// LS Electric XG5000 project: 16-48-1
// PLC NewPLC
// module base 0 slot 0: 입출력 모듈:XBC-DR14E (DC 24V 입력 8점, 릴레이 출력 6점)

PROGRAM NewProgram (task: 스캔 프로그램)

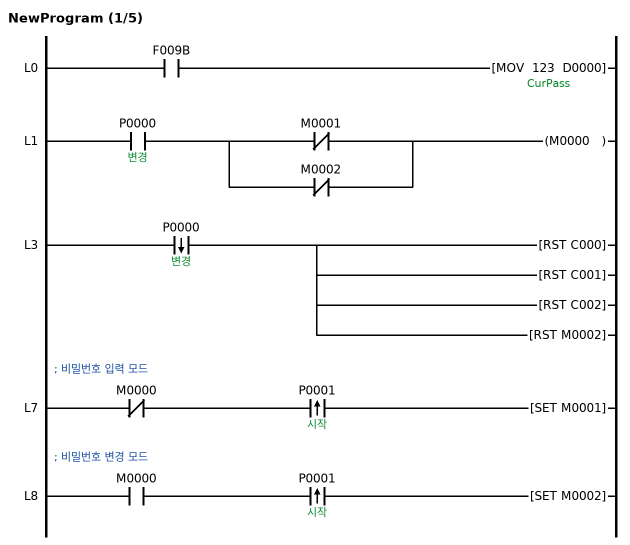
; L0
LOAD      F009B
MOV       123 D0000	// CurPass
; L1
LOAD      P0000	// 변경
LOAD NOT  M0001
OR NOT    M0002
AND LOAD
OUT       M0000
; L3
LOADN     P0000	// 변경
RST       C000
RST       C001
RST       C002
RST       M0002
; L7
LOAD NOT  M0000
ANDP      P0001	// 시작
SET       M0001
// output comment: 비밀번호 입력 모드
; L8
LOAD      M0000
ANDP      P0001	// 시작
SET       M0002
// output comment: 비밀번호 변경 모드

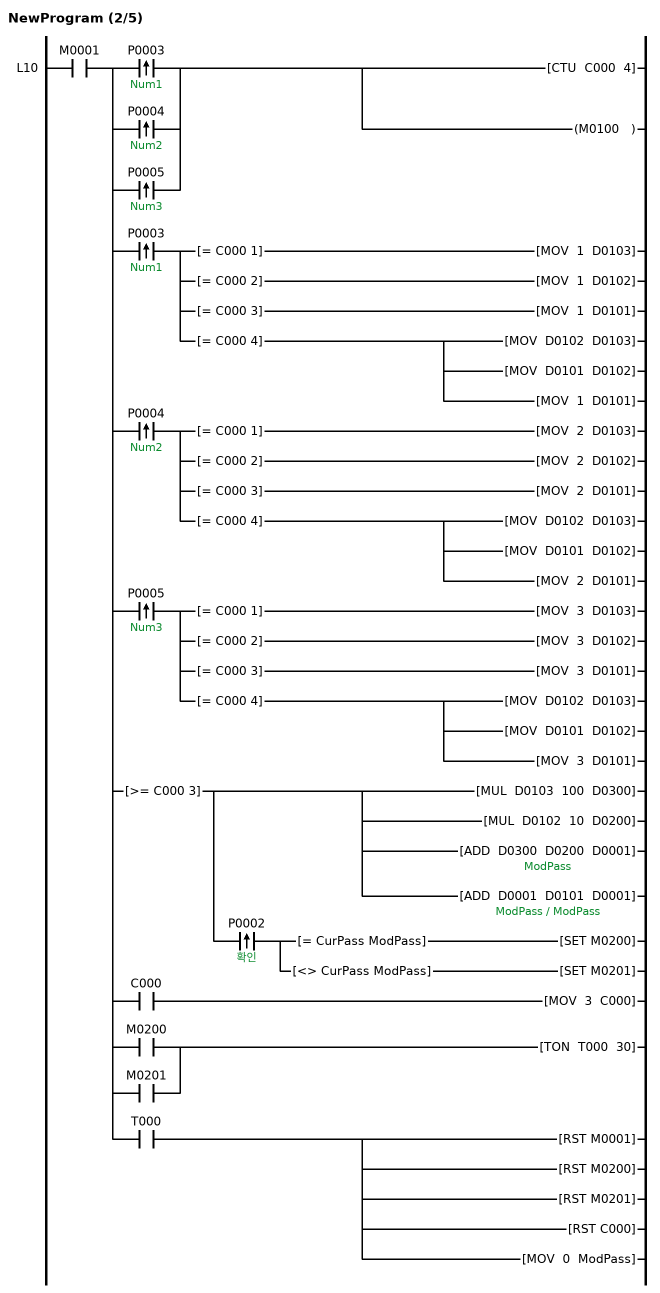
; L10
LOAD      M0001
MPUSH
LOADP     P0003	// Num1
ORP       P0004	// Num2
ORP       P0005	// Num3
AND LOAD
CTU       C000 4
OUT       M0100
MLOAD
ANDP      P0003	// Num1
MPUSH
AND=      C000 1
MOV       1 D0103
MLOAD
AND=      C000 2
MOV       1 D0102
MLOAD
AND=      C000 3
MOV       1 D0101
MPOP
AND=      C000 4
MOV       D0102 D0103
MOV       D0101 D0102
MOV       1 D0101
MLOAD
ANDP      P0004	// Num2
MPUSH
AND=      C000 1
MOV       2 D0103
MLOAD
AND=      C000 2
MOV       2 D0102
MLOAD
AND=      C000 3
MOV       2 D0101
MPOP
AND=      C000 4
MOV       D0102 D0103
MOV       D0101 D0102
MOV       2 D0101
MLOAD
ANDP      P0005	// Num3
MPUSH
AND=      C000 1
MOV       3 D0103
MLOAD
AND=      C000 2
MOV       3 D0102
MLOAD
AND=      C000 3
MOV       3 D0101
MPOP
AND=      C000 4
MOV       D0102 D0103
MOV       D0101 D0102
MOV       3 D0101
MLOAD
AND>=     C000 3
MUL       D0103 100 D0300
MUL       D0102 10 D0200
ADD       D0300 D0200 D0001	// ModPass
ADD       D0001 D0101 D0001	// ModPass / ModPass
ANDP      P0002	// 확인
MPUSH
AND=      CurPass ModPass
SET       M0200
MPOP
AND<>     CurPass ModPass
SET       M0201
MLOAD
AND       C000
MOV       3 C000
MLOAD
LOAD      M0200
OR        M0201
AND LOAD
TON       T000 30
MPOP
AND       T000
RST       M0001
RST       M0200
RST       M0201
RST       C000
MOV       0 ModPass

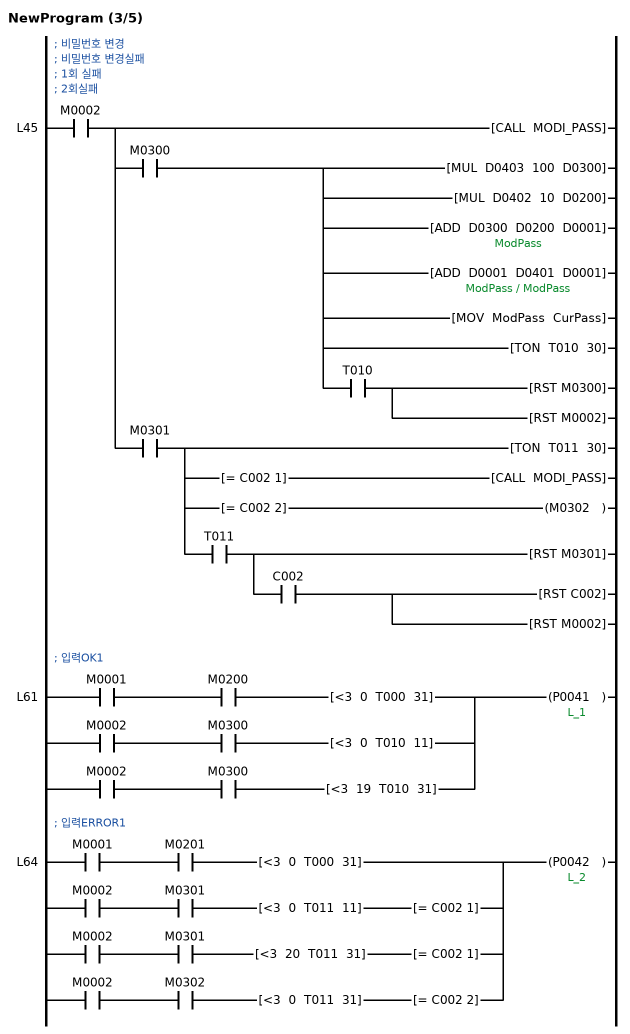
; L45
LOAD      M0002
CALL      MODI_PASS
MPUSH
AND       M0300
MUL       D0403 100 D0300
MUL       D0402 10 D0200
ADD       D0300 D0200 D0001	// ModPass
ADD       D0001 D0401 D0001	// ModPass / ModPass
MOV       ModPass CurPass
TON       T010 30
AND       T010
RST       M0300
RST       M0002
MPOP
AND       M0301
TON       T011 30
MPUSH
AND=      C002 1
CALL      MODI_PASS
MLOAD
AND=      C002 2
OUT       M0302
MPOP
AND       T011
RST       M0301
AND       C002
RST       C002
RST       M0002
// output comment: 비밀번호 변경
// output comment: 비밀번호 변경실패
// output comment: 1회 실패
// output comment: 2회실패
; L61
LOAD      M0001
AND       M0200
AND<3     0 T000 31
LOAD      M0002
AND       M0300
AND<3     0 T010 11
OR LOAD
LOAD      M0002
AND       M0300
AND<3     19 T010 31
OR LOAD
OUT       P0041	// L_1
// output comment: 입력OK1
; L64
LOAD      M0001
AND       M0201
AND<3     0 T000 31
LOAD      M0002
AND       M0301
AND<3     0 T011 11
AND=      C002 1
OR LOAD
LOAD      M0002
AND       M0301
AND<3     20 T011 31
AND=      C002 1
OR LOAD
LOAD      M0002
AND       M0302
AND<3     0 T011 31
AND=      C002 2
OR LOAD
OUT       P0042	// L_2
// output comment: 입력ERROR1

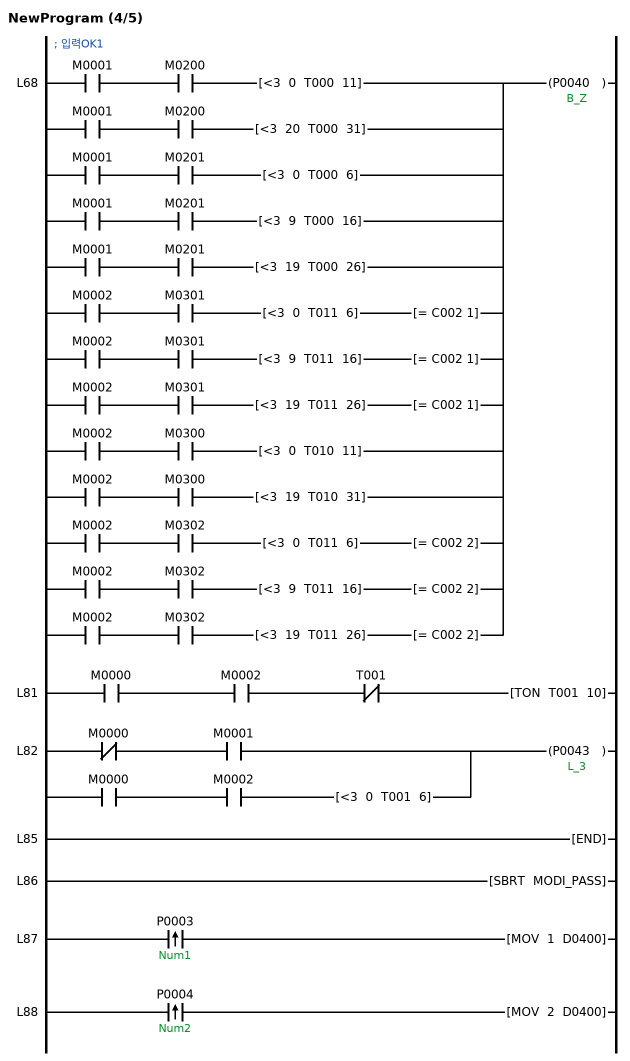
; L68
LOAD      M0001
AND       M0200
AND<3     0 T000 11
LOAD      M0001
AND       M0200
AND<3     20 T000 31
OR LOAD
LOAD      M0001
AND       M0201
AND<3     0 T000 6
OR LOAD
LOAD      M0001
AND       M0201
AND<3     9 T000 16
OR LOAD
LOAD      M0001
AND       M0201
AND<3     19 T000 26
OR LOAD
LOAD      M0002
AND       M0301
AND<3     0 T011 6
AND=      C002 1
OR LOAD
LOAD      M0002
AND       M0301
AND<3     9 T011 16
AND=      C002 1
OR LOAD
LOAD      M0002
AND       M0301
AND<3     19 T011 26
AND=      C002 1
OR LOAD
LOAD      M0002
AND       M0300
AND<3     0 T010 11
OR LOAD
LOAD      M0002
AND       M0300
AND<3     19 T010 31
OR LOAD
LOAD      M0002
AND       M0302
AND<3     0 T011 6
AND=      C002 2
OR LOAD
LOAD      M0002
AND       M0302
AND<3     9 T011 16
AND=      C002 2
OR LOAD
LOAD      M0002
AND       M0302
AND<3     19 T011 26
AND=      C002 2
OR LOAD
OUT       P0040	// B_Z
// output comment: 입력OK1
; L81
LOAD      M0000
AND       M0002
AND NOT   T001
TON       T001 10
; L82
LOAD NOT  M0000
AND       M0001
LOAD      M0000
AND       M0002
AND<3     0 T001 6
OR LOAD
OUT       P0043	// L_3
; L85
END
; L86
SBRT      MODI_PASS
; L87
LOADP     P0003	// Num1
MOV       1 D0400
; L88
LOADP     P0004	// Num2
MOV       2 D0400

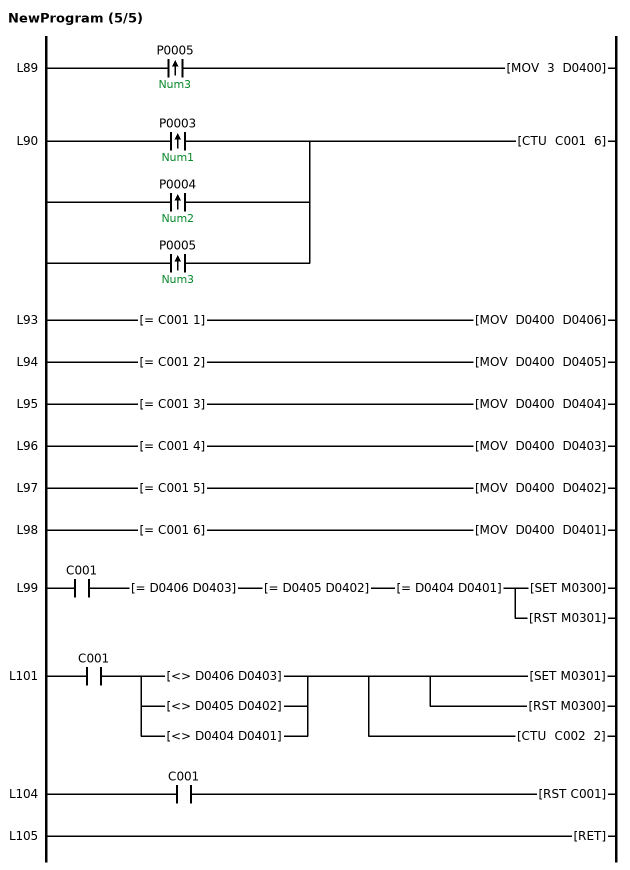
; L89
LOADP     P0005	// Num3
MOV       3 D0400
; L90
LOADP     P0003	// Num1
ORP       P0004	// Num2
ORP       P0005	// Num3
CTU       C001 6
; L93
LOAD=     C001 1
MOV       D0400 D0406
; L94
LOAD=     C001 2
MOV       D0400 D0405
; L95
LOAD=     C001 3
MOV       D0400 D0404
; L96
LOAD=     C001 4
MOV       D0400 D0403
; L97
LOAD=     C001 5
MOV       D0400 D0402
; L98
LOAD=     C001 6
MOV       D0400 D0401
; L99
LOAD      C001
AND=      D0406 D0403
AND=      D0405 D0402
AND=      D0404 D0401
SET       M0300
RST       M0301
; L101
LOAD      C001
LOAD<>    D0406 D0403
OR<>      D0405 D0402
OR<>      D0404 D0401
AND LOAD
SET       M0301
RST       M0300
CTU       C002 2
; L104
LOAD      C001
RST       C001
; L105
RET